TYPE ST_General_LeakTester :
STRUCT
	
	sti28General_I_O					: st_i28General_I_O;
	sti28LasResult						: st_i28LasResult;
	sti28LiveMeasurement				: st_i28LiveMeasurement;

END_STRUCT
END_TYPE

(* stored: Version 1.1.0.1, ProductVersion 3.1.4024.13
   DUT ST_General_LeakTester: Id {cce0cedf-49f9-4006-a73b-4ed8a3a5a71d} *)
